PROGRAM P_Demo_FB_ReadDriveInfo
VAR
    fbReadInfo   : FB_ReadDriveInfo; // 读驱动器信息 FB 实例
    axisMain     : AXIS_REF; // 主轴轴引用；必须先在 System Manager 配好并 Link
    rtReadTrig   : R_TRIG; // 把电平转上升沿
    bReadInfoReq : BOOL := FALSE; // 在线写 TRUE 触发一次读取
    stDriveInfo  : ST_DriveInfo; // 读回的驱动器寻址信息；Done 后有效
    bInfoDone    : BOOL;
    bInfoBusy    : BOOL;
    bInfoError   : BOOL;
    nInfoErrorID : UDINT;
END_VAR

// =============================================================================
// 场景：设备初始化阶段，从 NC 轴自动读出所连驱动器的 NetId / 从站地址 /
//       设备类型，供后续 FB_SoERead / FB_CoERead 访问参数时使用，避免在
//       代码里写死从站寻址信息。
//
// 价值：1) 代码不写死 NetId / SlaveAddress，跟着 System Manager 配置走
//       2) 本 FB 有 Done 输出，Done 上升沿即"DriveInfo 就绪"，最直观
//       3) DeviceType 可用于分支不同型号（SoE vs CoE）的逻辑
//
// 验证步骤：
//   1. System Manager 配好 NC 轴并 Link 给 axisMain，引用 Tc2_MC2_Drive
//   2. Add Existing Item (.TcPOU) 选本文件，加进 PlcTask，编译登录
//   3. 在线写 bReadInfoReq := TRUE → bInfoBusy 置 TRUE
//   4. 等 bInfoDone 置 TRUE → 展开 stDriveInfo 应看到 NetId / SlaveAddress /
//      DeviceName / DeviceType 等字段被填上有效值
//   5. 若 bInfoError = TRUE，看 nInfoErrorID 对照 ADS Return Codes 表
//   6. 把 bReadInfoReq 拉回 FALSE 复位边沿；配置不变时初始化读一次即可
// =============================================================================

// 用 R_TRIG 把"持续按住的 TRUE"转成真正的上升沿
rtReadTrig(CLK := bReadInfoReq);

// 单次调用：本 FB 有 Done 输出，Axis 是 VAR_IN_OUT 必传
fbReadInfo(
    Execute   := rtReadTrig.Q,
    Axis      := axisMain,
    Done      => bInfoDone,
    Busy      => bInfoBusy,
    Error     => bInfoError,
    ErrorID   => nInfoErrorID,
    DriveInfo => stDriveInfo
);

END_PROGRAM

(* stored: Version 1.1.0.1, ProductVersion 3.1.4024.5
   POU P_Demo_FB_ReadDriveInfo: Id {d7afc1e4-ca91-5510-88e8-549cece44c69}, SpecialFunc None *)
